TYPE S_SkyCoordHorizontal :
STRUCT
	alt:	LREAL;
	az:		LREAL;
END_STRUCT
END_TYPE

(* stored: Version 1.1.0.1, ProductVersion 3.1.4024.12
   DUT S_SkyCoordHorizontal: Id {bc934920-5c3a-495a-b2a3-4fcfc22f927a} *)
